INTERFACE ITcoMessengerSettings

PROPERTY IsSuspended : BOOL
GET
END_GET
END_PROPERTY

PROPERTY MessageDigestMethod : eMessageDigestMethod
GET
END_GET
SET
END_SET
END_PROPERTY

PROPERTY MessengerLoggingMethod : eMessengerLogMethod
GET
END_GET
SET
END_SET
END_PROPERTY

PROPERTY MinLevel : eMessageCategory
GET
END_GET
SET
END_SET
END_PROPERTY

METHOD Resume : BOOL
VAR_INPUT
END_VAR
END_METHOD

METHOD Suspend
END_METHOD

END_INTERFACE

(* stored: Version 1.1.0.1
   Itf ITcoMessengerSettings: Id {6d6b9064-8fe9-0b02-00be-c0f0ff54eeb4}
   Property IsSuspended: Id {154b3f83-5ad6-0af7-30ee-bb7fbba61c91}
   Get Get: Id {f4387df2-7158-0155-1a2d-255a7974d7ab}
   Property MessageDigestMethod: Id {7a7aeee6-0c64-0e00-156f-dfaae334f461}
   Get Get: Id {34e87f8f-f513-0ad8-07a5-140cc54b9bfb}
   Set Set: Id {e8c02ca8-9667-046a-024f-887a88359d43}
   Property MessengerLoggingMethod: Id {cfc43eb5-278e-0822-2269-dbd2e76dc73a}
   Get Get: Id {1904dd58-ebb4-0664-0201-aac49e6e4696}
   Set Set: Id {f8a21ff8-7f65-0940-0f4b-d0c8ca94a71c}
   Property MinLevel: Id {affff53c-8111-0dde-30b4-02bee538a109}
   Get Get: Id {229f0b50-4658-067e-0200-914aca38739d}
   Set Set: Id {39ad8fc0-c4c1-0ff8-112c-8be3a37d8762}
   Method Resume: Id {7e5e1860-858e-0160-39b2-f7bfc3ac189a}
   Method Suspend: Id {d170a192-4a15-0a78-14b9-e61ea3ece139} *)
